// TIA Portal V16 export
// export: Created 2022-09-01T13:37:22.0100117Z, ExportSetting WithDefaults, DisplayName Totally Integrated Automation Portal, DisplayVersion V16, DisplayName TIA Portal Version Control Interface, DisplayVersion V16, DisplayName TIA Portal Openness, DisplayVersion V16, DisplayName STEP 7 Professional, DisplayVersion V16, DisplayName STEP 7 Safety, DisplayVersion V16, DisplayName WinCC Advanced, DisplayVersion V16
VAR_GLOBAL   // PLC tag table "Default tag table"
   FirstScan AT %M1.0 : Bool;
   FALLING_EDGE_MAN_AUTO AT %M100.0 : Bool;
   RISING_EDGE_ETAPA_6 AT %M100.2 : Bool;
   FALLING_EDGE_BOT_EMERG AT %M100.5 : Bool;
   FALLIN_EDGE_BOT_EMERG_2 AT %M100.6 : Bool;
   FALLING_EDGE_ETAPA_6 AT %M100.7 : Bool;
   MBIT_DISP_1 AT %M101.0 : Bool;
   MBIT_DISP_2 AT %M101.1 : Bool;
   MBIT_DISP_3 AT %M101.2 : Bool;
   MBIT_DISP_4 AT %M101.3 : Bool;
   MBIT_DISP_5 AT %M101.4 : Bool;
   MBIT_DISP_6 AT %M101.5 : Bool;
   MBIT_DISP_7 AT %M101.6 : Bool;
   MBIT_DISP_8 AT %M101.7 : Bool;
   MBIT_DISP_9 AT %M102.0 : Bool;
   MBIT_DISP_10 AT %M102.1 : Bool;
   MBIT_DISP_11 AT %M102.2 : Bool;
   MBIT_DISP_12 AT %M102.3 : Bool;
   MBIT_DISP_13 AT %M102.4 : Bool;
   MBIT_DISP_14 AT %M102.5 : Bool;
   MBIT_DISP_15 AT %M102.6 : Bool;
   MBIT_DISP_16 AT %M102.7 : Bool;
   MBIT_DISP_DIF_3Q1_32 AT %M103.0 : Bool;
   MBIT_DISP_DIF_3Q3 AT %M103.1 : Bool;
   MBIT_DISP_DIF_4Q1_4Q2 AT %M103.2 : Bool;
   MBIT_FALHA_24VDC AT %M103.3 : Bool;
   MBIT_FALHA_220VAC AT %M103.4 : Bool;
   MBIT_FALHA_24VAC AT %M103.5 : Bool;
   RISING_EDGE_ETAPA_55 AT %M103.7 : Bool;
   RISING_EDGE_START_CICLO AT %M104.0 : Bool;
   Tag_1 AT %M200.0 : Bool;
END_VAR
